FUNCTION_BLOCK SREAMING_PLOT_4_TIMESERIES
  {SET_ATTRIBUTE(OpcUa, SERVICE)}
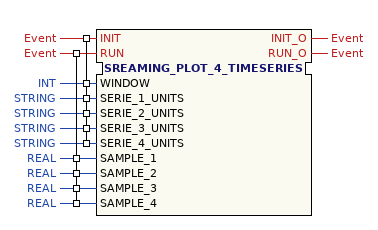
  EVENT_INPUT
    INIT WITH WINDOW, SERIE_1_UNITS, SERIE_2_UNITS, SERIE_3_UNITS, SERIE_4_UNITS;
    RUN WITH SAMPLE_1, SAMPLE_2, SAMPLE_3, SAMPLE_4;
  END_EVENT
  EVENT_OUTPUT
    INIT_O;
    RUN_O;
  END_EVENT
  VAR_INPUT
    WINDOW : INT; {SET_ATTRIBUTE(OpcUa, Constant.RUN)}
    SERIE_1_UNITS : STRING; {SET_ATTRIBUTE(OpcUa, Constant.RUN)}
    SERIE_2_UNITS : STRING; {SET_ATTRIBUTE(OpcUa, Constant.RUN)}
    SERIE_3_UNITS : STRING; {SET_ATTRIBUTE(OpcUa, Constant.RUN)}
    SERIE_4_UNITS : STRING; {SET_ATTRIBUTE(OpcUa, Constant.RUN)}
    SAMPLE_1 : REAL; {SET_ATTRIBUTE(OpcUa, Variable.RUN)}
    SAMPLE_2 : REAL; {SET_ATTRIBUTE(OpcUa, Variable.RUN)}
    SAMPLE_3 : REAL; {SET_ATTRIBUTE(OpcUa, Variable.RUN)}
    SAMPLE_4 : REAL; {SET_ATTRIBUTE(OpcUa, Variable.RUN)}
  END_VAR
END_FUNCTION_BLOCK
